PROGRAM MAIN
VAR
	
END_VAR


POU_Seguridad();
POU_Mando();
POU_Funcionamiento();

END_PROGRAM

(* stored: Version 1.1.0.1, ProductVersion 3.1.4024.12
   POU MAIN: Id {7ad81a30-7aa4-44e3-9151-5703448cad9a}, SpecialFunc None *)
